// TIA Portal V17 export
// export: Created 2023-03-06T02:05:12.3050921Z, ExportSetting WithDefaults, DisplayName Totally Integrated Automation Portal, DisplayVersion V17 Update 4, DisplayName TIA Portal Openness, DisplayVersion V17 Update 4, DisplayName TIA Portal Version Control Interface, DisplayVersion V17, DisplayName STEP 7 Professional, DisplayVersion V17 Update 4, DisplayName STEP 7 Safety, DisplayVersion V17, DisplayName WinCC Professional, DisplayVersion V17 Update 4
FUNCTION "PCS1 W (PE)" : Void   // FC42, LAD
TITLE = ModBus TCP for PCS Power Electronics
{ S7_Optimized_Access := 'TRUE' }
VERSION : 0.1
// stored: AutoNumber false, IsIECCheckEnabled false, SetENOAutomatically false, UDAEnableTagReadback false
   VAR_TEMP
      rSS1PacRef : Real;
      rSS2PacRef : Real;
      rSS1QacRef : Real;
      rSS2QacRef : Real;
      rSnHalfPE : Real;
   END_VAR
   VAR_TEMP   // added for the SCL form of the ladder/FBD networks
      _w1 : Bool;
      _w2 : Bool;
   END_VAR
BEGIN

REGION Network 1: Function Modbus Client
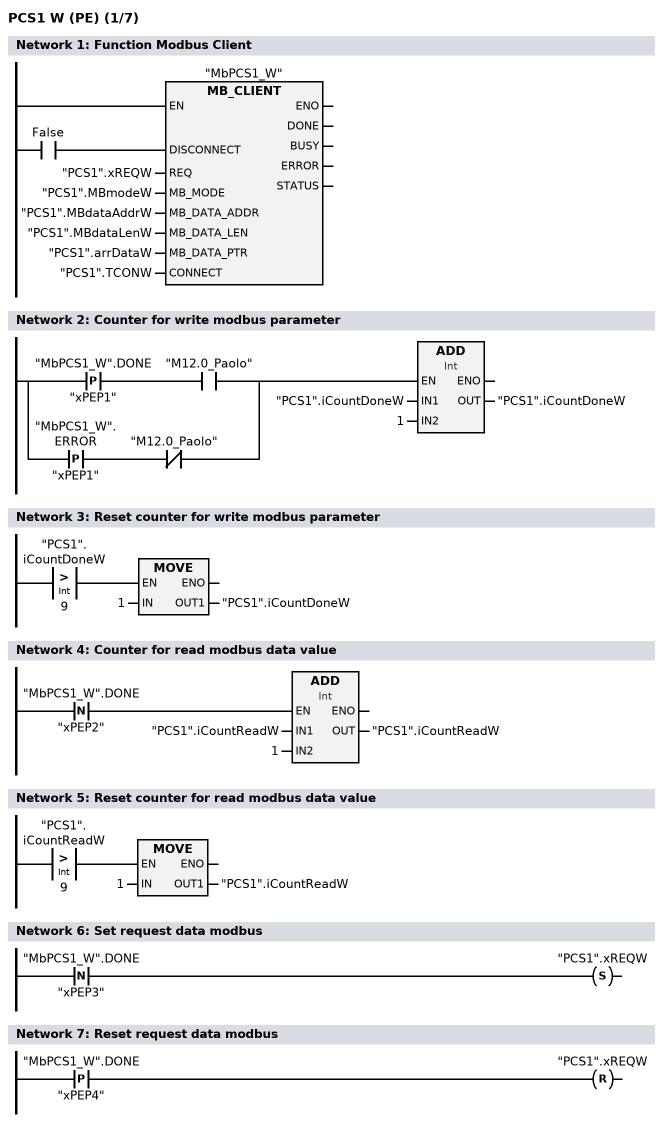
   RUNG wire#powerrail
      "MbPCS1_W".MB_CLIENT(DISCONNECT := wire#w1, REQ := "PCS1".xREQW, MB_MODE := "PCS1".MBmodeW, MB_DATA_ADDR := "PCS1".MBdataAddrW, MB_DATA_LEN := "PCS1".MBdataLenW, MB_DATA_PTR := "PCS1".arrDataW, CONNECT := "PCS1".TCONW, DONE =>, BUSY =>, ERROR =>, STATUS =>)
   END_RUNG
   RUNG wire#powerrail
      Contact( False )
   END_RUNG wire#w1
   // the same network as SCL:
   "MbPCS1_W"(DISCONNECT := False,   // MB_CLIENT
              REQ := "PCS1".xREQW,
              MB_MODE := "PCS1".MBmodeW,
              MB_DATA_ADDR := "PCS1".MBdataAddrW,
              MB_DATA_LEN := "PCS1".MBdataLenW,
              MB_DATA_PTR := "PCS1".arrDataW,
              CONNECT := "PCS1".TCONW);
END_REGION

REGION Network 2: Counter for write modbus parameter
   RUNG wire#powerrail
      P_Contact(operand := "MbPCS1_W".DONE, bit := "xPEP1")
      Contact( "M12.0_Paolo" )
      wire#w1
      { S7_Templates := "SrcType := Int" } Add(in1 := "PCS1".iCountDoneW, in2 := 1, out => "PCS1".iCountDoneW)
   END_RUNG
   RUNG wire#powerrail
      P_Contact(operand := "MbPCS1_W".ERROR, bit := "xPEP1")
      I_Contact( "M12.0_Paolo" )
   END_RUNG wire#w1
   // the same network as SCL:
   #_w1 := "MbPCS1_W".DONE AND NOT "xPEP1";   // rising edge of "MbPCS1_W".DONE
   "xPEP1" := "MbPCS1_W".DONE;
   #_w2 := "MbPCS1_W".ERROR AND NOT "xPEP1";   // rising edge of "MbPCS1_W".ERROR
   "xPEP1" := "MbPCS1_W".ERROR;
   IF (#_w1 AND "M12.0_Paolo") OR (#_w2 AND NOT "M12.0_Paolo") THEN
       "PCS1".iCountDoneW := "PCS1".iCountDoneW + 1;
   END_IF;
END_REGION

REGION Network 3: Reset counter for write modbus parameter
   RUNG wire#powerrail
      { S7_Templates := "SrcType := Int" } GT_Contact(in1 := "PCS1".iCountDoneW, in2 := 9)
      Move(in := 1, out1 => "PCS1".iCountDoneW)
   END_RUNG
   // the same network as SCL:
   IF "PCS1".iCountDoneW > 9 THEN "PCS1".iCountDoneW := 1; END_IF;
END_REGION

REGION Network 4: Counter for read modbus data value
   RUNG wire#powerrail
      N_Contact(operand := "MbPCS1_W".DONE, bit := "xPEP2")
      { S7_Templates := "SrcType := Int" } Add(in1 := "PCS1".iCountReadW, in2 := 1, out => "PCS1".iCountReadW)
   END_RUNG
   // the same network as SCL:
   #_w1 := NOT "MbPCS1_W".DONE AND "xPEP2";   // falling edge of "MbPCS1_W".DONE
   "xPEP2" := "MbPCS1_W".DONE;
   IF #_w1 THEN "PCS1".iCountReadW := "PCS1".iCountReadW + 1; END_IF;
END_REGION

REGION Network 5: Reset counter for read modbus data value
   RUNG wire#powerrail
      { S7_Templates := "SrcType := Int" } GT_Contact(in1 := "PCS1".iCountReadW, in2 := 9)
      Move(in := 1, out1 => "PCS1".iCountReadW)
   END_RUNG
   // the same network as SCL:
   IF "PCS1".iCountReadW > 9 THEN "PCS1".iCountReadW := 1; END_IF;
END_REGION

REGION Network 6: Set request data modbus
   RUNG wire#powerrail
      N_Contact(operand := "MbPCS1_W".DONE, bit := "xPEP3")
      S_Coil( "PCS1".xREQW )
   END_RUNG
   // the same network as SCL:
   #_w1 := NOT "MbPCS1_W".DONE AND "xPEP3";   // falling edge of "MbPCS1_W".DONE
   "xPEP3" := "MbPCS1_W".DONE;
   IF #_w1 THEN "PCS1".xREQW := TRUE; END_IF;
END_REGION

REGION Network 7: Reset request data modbus
   RUNG wire#powerrail
      P_Contact(operand := "MbPCS1_W".DONE, bit := "xPEP4")
      R_Coil( "PCS1".xREQW )
   END_RUNG
   // the same network as SCL:
   #_w1 := "MbPCS1_W".DONE AND NOT "xPEP4";   // rising edge of "MbPCS1_W".DONE
   "xPEP4" := "MbPCS1_W".DONE;
   IF #_w1 THEN "PCS1".xREQW := FALSE; END_IF;
END_REGION

REGION Network 9: Write W_Block1 parameter
   // wUserPswIns
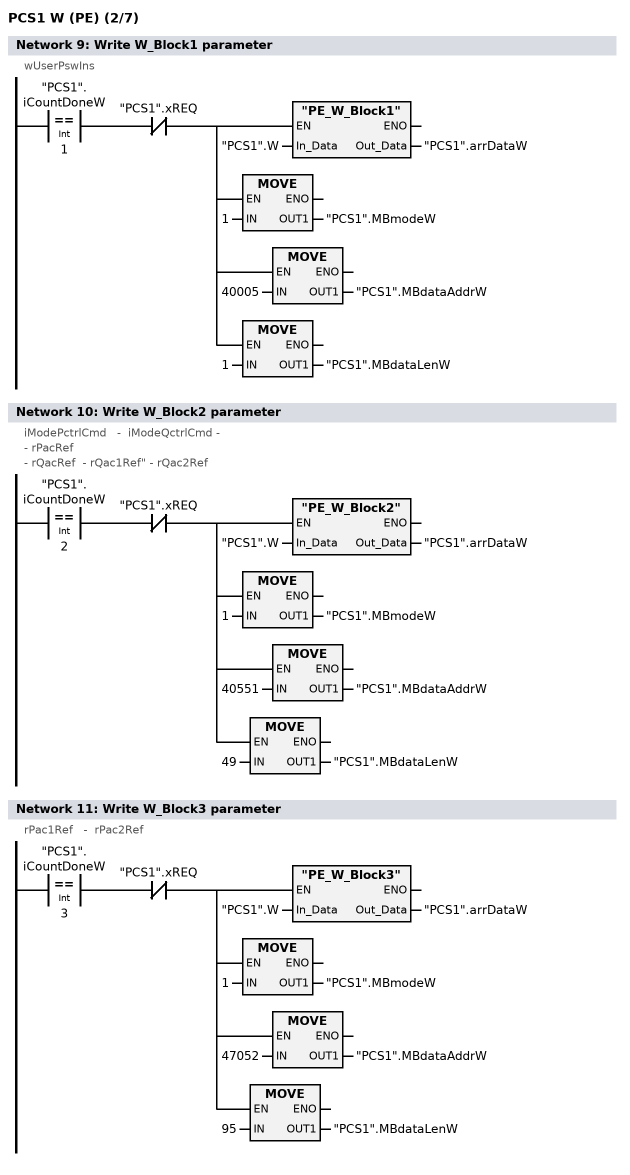
   RUNG wire#powerrail
      { S7_Templates := "SrcType := Int" } EQ_Contact(in1 := "PCS1".iCountDoneW, in2 := 1)
      I_Contact( "PCS1".xREQ )
      wire#w1
      "PE_W_Block1"(In_Data := "PCS1".W, Out_Data => "PCS1".arrDataW)
   END_RUNG
   RUNG wire#w1
      Move(in := 1, out1 => "PCS1".MBmodeW)
   END_RUNG
   RUNG wire#w1
      Move(in := 40005, out1 => "PCS1".MBdataAddrW)
   END_RUNG
   RUNG wire#w1
      Move(in := 1, out1 => "PCS1".MBdataLenW)
   END_RUNG
   // the same network as SCL:
   #_w1 := ("PCS1".iCountDoneW = 1) AND NOT "PCS1".xREQ;
   IF #_w1 THEN
       "PE_W_Block1"(In_Data := "PCS1".W, Out_Data => "PCS1".arrDataW);
       "PCS1".MBmodeW := 1;
       "PCS1".MBdataAddrW := 40005;
       "PCS1".MBdataLenW := 1;
   END_IF;
END_REGION

REGION Network 10: Write W_Block2 parameter
   // iModePctrlCmd   -  iModeQctrlCmd - 
   // - rPacRef 
   // - rQacRef  - rQac1Ref" - rQac2Ref
   RUNG wire#powerrail
      { S7_Templates := "SrcType := Int" } EQ_Contact(in1 := "PCS1".iCountDoneW, in2 := 2)
      I_Contact( "PCS1".xREQ )
      wire#w1
      "PE_W_Block2"(In_Data := "PCS1".W, Out_Data => "PCS1".arrDataW)
   END_RUNG
   RUNG wire#w1
      Move(in := 1, out1 => "PCS1".MBmodeW)
   END_RUNG
   RUNG wire#w1
      Move(in := 40551, out1 => "PCS1".MBdataAddrW)
   END_RUNG
   RUNG wire#w1
      Move(in := 49, out1 => "PCS1".MBdataLenW)
   END_RUNG
   // the same network as SCL:
   #_w1 := ("PCS1".iCountDoneW = 2) AND NOT "PCS1".xREQ;
   IF #_w1 THEN
       "PE_W_Block2"(In_Data := "PCS1".W, Out_Data => "PCS1".arrDataW);
       "PCS1".MBmodeW := 1;
       "PCS1".MBdataAddrW := 40551;
       "PCS1".MBdataLenW := 49;
   END_IF;
END_REGION

REGION Network 11: Write W_Block3 parameter
   // rPac1Ref   -  rPac2Ref
   RUNG wire#powerrail
      { S7_Templates := "SrcType := Int" } EQ_Contact(in1 := "PCS1".iCountDoneW, in2 := 3)
      I_Contact( "PCS1".xREQ )
      wire#w1
      "PE_W_Block3"(In_Data := "PCS1".W, Out_Data => "PCS1".arrDataW)
   END_RUNG
   RUNG wire#w1
      Move(in := 1, out1 => "PCS1".MBmodeW)
   END_RUNG
   RUNG wire#w1
      Move(in := 47052, out1 => "PCS1".MBdataAddrW)
   END_RUNG
   RUNG wire#w1
      Move(in := 95, out1 => "PCS1".MBdataLenW)
   END_RUNG
   // the same network as SCL:
   #_w1 := ("PCS1".iCountDoneW = 3) AND NOT "PCS1".xREQ;
   IF #_w1 THEN
       "PE_W_Block3"(In_Data := "PCS1".W, Out_Data => "PCS1".arrDataW);
       "PCS1".MBmodeW := 1;
       "PCS1".MBdataAddrW := 47052;
       "PCS1".MBdataLenW := 95;
   END_IF;
END_REGION

REGION Network 12: Write Command Start
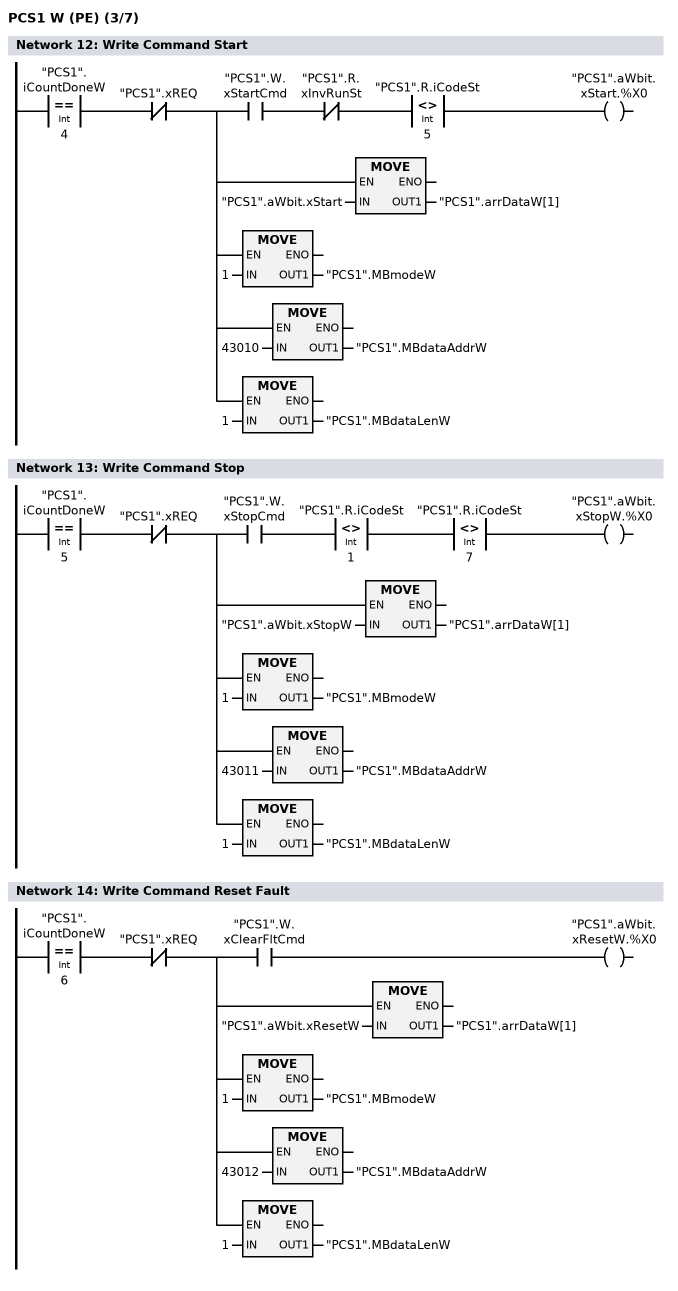
   RUNG wire#powerrail
      { S7_Templates := "SrcType := Int" } EQ_Contact(in1 := "PCS1".iCountDoneW, in2 := 4)
      I_Contact( "PCS1".xREQ )
      wire#w1
      Contact( "PCS1".W.xStartCmd )
      I_Contact( "PCS1".R.xInvRunSt )
      { S7_Templates := "SrcType := Int" } NE_Contact(in1 := "PCS1".R.iCodeSt, in2 := 5)
      Coil( "PCS1".aWbit.xStart.%X0 )
   END_RUNG
   RUNG wire#w1
      Move(in := "PCS1".aWbit.xStart, out1 => "PCS1".arrDataW[1])
   END_RUNG
   RUNG wire#w1
      Move(in := 1, out1 => "PCS1".MBmodeW)
   END_RUNG
   RUNG wire#w1
      Move(in := 43010, out1 => "PCS1".MBdataAddrW)
   END_RUNG
   RUNG wire#w1
      Move(in := 1, out1 => "PCS1".MBdataLenW)
   END_RUNG
   // the same network as SCL:
   #_w1 := ("PCS1".iCountDoneW = 4) AND NOT "PCS1".xREQ;
   "PCS1".aWbit.xStart.%X0 := #_w1 AND "PCS1".W.xStartCmd AND NOT "PCS1".R.xInvRunSt AND ("PCS1".R.iCodeSt <> 5);
   IF #_w1 THEN
       "PCS1".arrDataW[1] := "PCS1".aWbit.xStart;
       "PCS1".MBmodeW := 1;
       "PCS1".MBdataAddrW := 43010;
       "PCS1".MBdataLenW := 1;
   END_IF;
END_REGION

REGION Network 13: Write Command Stop
   RUNG wire#powerrail
      { S7_Templates := "SrcType := Int" } EQ_Contact(in1 := "PCS1".iCountDoneW, in2 := 5)
      I_Contact( "PCS1".xREQ )
      wire#w1
      Contact( "PCS1".W.xStopCmd )
      { S7_Templates := "SrcType := Int" } NE_Contact(in1 := "PCS1".R.iCodeSt, in2 := 1)
      { S7_Templates := "SrcType := Int" } NE_Contact(in1 := "PCS1".R.iCodeSt, in2 := 7)
      Coil( "PCS1".aWbit.xStopW.%X0 )
   END_RUNG
   RUNG wire#w1
      Move(in := "PCS1".aWbit.xStopW, out1 => "PCS1".arrDataW[1])
   END_RUNG
   RUNG wire#w1
      Move(in := 1, out1 => "PCS1".MBmodeW)
   END_RUNG
   RUNG wire#w1
      Move(in := 43011, out1 => "PCS1".MBdataAddrW)
   END_RUNG
   RUNG wire#w1
      Move(in := 1, out1 => "PCS1".MBdataLenW)
   END_RUNG
   // the same network as SCL:
   #_w1 := ("PCS1".iCountDoneW = 5) AND NOT "PCS1".xREQ;
   "PCS1".aWbit.xStopW.%X0 := #_w1 AND "PCS1".W.xStopCmd AND ("PCS1".R.iCodeSt <> 1) AND ("PCS1".R.iCodeSt <> 7);
   IF #_w1 THEN
       "PCS1".arrDataW[1] := "PCS1".aWbit.xStopW;
       "PCS1".MBmodeW := 1;
       "PCS1".MBdataAddrW := 43011;
       "PCS1".MBdataLenW := 1;
   END_IF;
END_REGION

REGION Network 14: Write Command Reset Fault
   RUNG wire#powerrail
      { S7_Templates := "SrcType := Int" } EQ_Contact(in1 := "PCS1".iCountDoneW, in2 := 6)
      I_Contact( "PCS1".xREQ )
      wire#w1
      Contact( "PCS1".W.xClearFltCmd )
      Coil( "PCS1".aWbit.xResetW.%X0 )
   END_RUNG
   RUNG wire#w1
      Move(in := "PCS1".aWbit.xResetW, out1 => "PCS1".arrDataW[1])
   END_RUNG
   RUNG wire#w1
      Move(in := 1, out1 => "PCS1".MBmodeW)
   END_RUNG
   RUNG wire#w1
      Move(in := 43012, out1 => "PCS1".MBdataAddrW)
   END_RUNG
   RUNG wire#w1
      Move(in := 1, out1 => "PCS1".MBdataLenW)
   END_RUNG
   // the same network as SCL:
   #_w1 := ("PCS1".iCountDoneW = 6) AND NOT "PCS1".xREQ;
   "PCS1".aWbit.xResetW.%X0 := #_w1 AND "PCS1".W.xClearFltCmd;
   IF #_w1 THEN
       "PCS1".arrDataW[1] := "PCS1".aWbit.xResetW;
       "PCS1".MBmodeW := 1;
       "PCS1".MBdataAddrW := 43012;
       "PCS1".MBdataLenW := 1;
   END_IF;
END_REGION

REGION Network 15: Write Command Enable Start/Stop
   // Con versione vecchia si usava solo questo registro per marcia ed arresto.
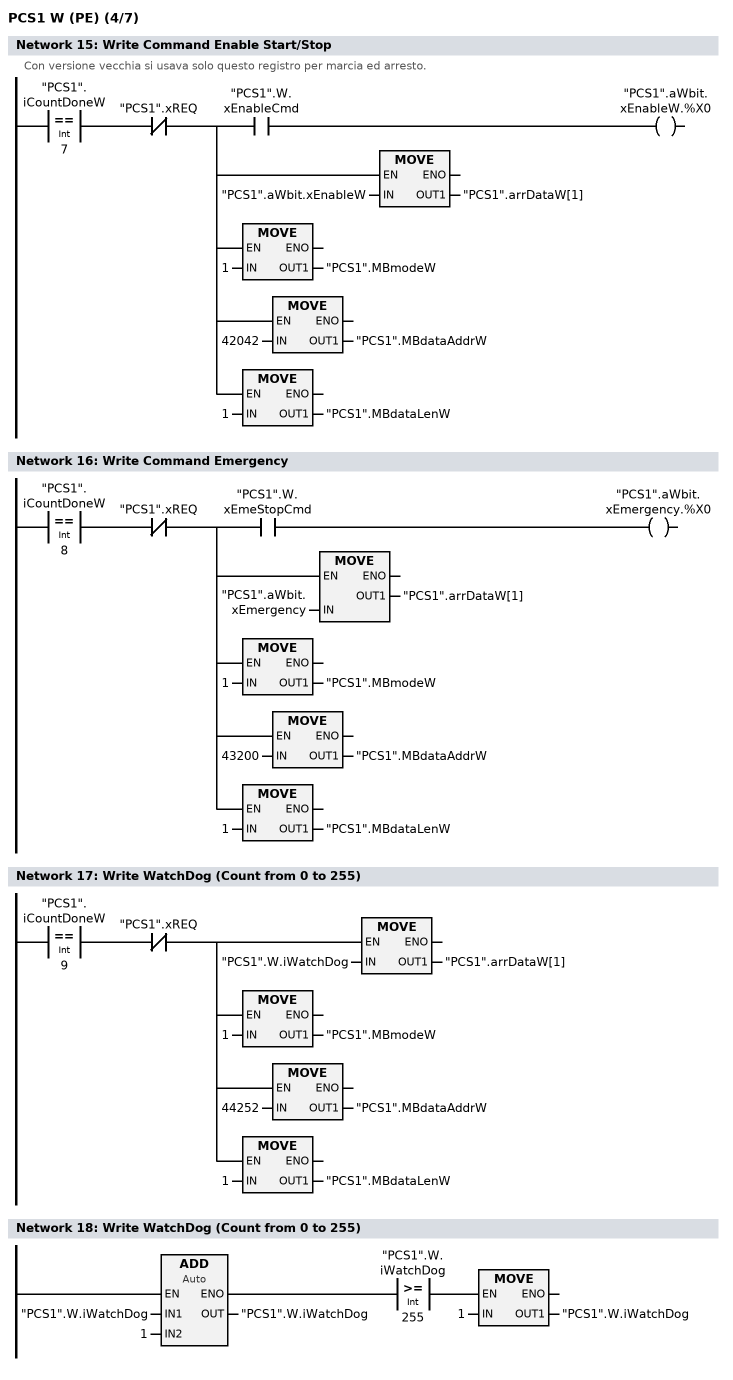
   RUNG wire#powerrail
      { S7_Templates := "SrcType := Int" } EQ_Contact(in1 := "PCS1".iCountDoneW, in2 := 7)
      I_Contact( "PCS1".xREQ )
      wire#w1
      Contact( "PCS1".W.xEnableCmd )
      Coil( "PCS1".aWbit.xEnableW.%X0 )
   END_RUNG
   RUNG wire#w1
      Move(in := "PCS1".aWbit.xEnableW, out1 => "PCS1".arrDataW[1])
   END_RUNG
   RUNG wire#w1
      Move(in := 1, out1 => "PCS1".MBmodeW)
   END_RUNG
   RUNG wire#w1
      Move(in := 42042, out1 => "PCS1".MBdataAddrW)
   END_RUNG
   RUNG wire#w1
      Move(in := 1, out1 => "PCS1".MBdataLenW)
   END_RUNG
   // the same network as SCL:
   #_w1 := ("PCS1".iCountDoneW = 7) AND NOT "PCS1".xREQ;
   "PCS1".aWbit.xEnableW.%X0 := #_w1 AND "PCS1".W.xEnableCmd;
   IF #_w1 THEN
       "PCS1".arrDataW[1] := "PCS1".aWbit.xEnableW;
       "PCS1".MBmodeW := 1;
       "PCS1".MBdataAddrW := 42042;
       "PCS1".MBdataLenW := 1;
   END_IF;
END_REGION

REGION Network 16: Write Command Emergency
   RUNG wire#powerrail
      { S7_Templates := "SrcType := Int" } EQ_Contact(in1 := "PCS1".iCountDoneW, in2 := 8)
      I_Contact( "PCS1".xREQ )
      wire#w1
      Contact( "PCS1".W.xEmeStopCmd )
      Coil( "PCS1".aWbit.xEmergency.%X0 )
   END_RUNG
   RUNG wire#w1
      Move(in := "PCS1".aWbit.xEmergency, out1 => "PCS1".arrDataW[1])
   END_RUNG
   RUNG wire#w1
      Move(in := 1, out1 => "PCS1".MBmodeW)
   END_RUNG
   RUNG wire#w1
      Move(in := 43200, out1 => "PCS1".MBdataAddrW)
   END_RUNG
   RUNG wire#w1
      Move(in := 1, out1 => "PCS1".MBdataLenW)
   END_RUNG
   // the same network as SCL:
   #_w1 := ("PCS1".iCountDoneW = 8) AND NOT "PCS1".xREQ;
   "PCS1".aWbit.xEmergency.%X0 := #_w1 AND "PCS1".W.xEmeStopCmd;
   IF #_w1 THEN
       "PCS1".arrDataW[1] := "PCS1".aWbit.xEmergency;
       "PCS1".MBmodeW := 1;
       "PCS1".MBdataAddrW := 43200;
       "PCS1".MBdataLenW := 1;
   END_IF;
END_REGION

REGION Network 17: Write WatchDog (Count from 0 to 255)
   RUNG wire#powerrail
      { S7_Templates := "SrcType := Int" } EQ_Contact(in1 := "PCS1".iCountDoneW, in2 := 9)
      I_Contact( "PCS1".xREQ )
      wire#w1
      Move(in := "PCS1".W.iWatchDog, out1 => "PCS1".arrDataW[1])
   END_RUNG
   RUNG wire#w1
      Move(in := 1, out1 => "PCS1".MBmodeW)
   END_RUNG
   RUNG wire#w1
      Move(in := 44252, out1 => "PCS1".MBdataAddrW)
   END_RUNG
   RUNG wire#w1
      Move(in := 1, out1 => "PCS1".MBdataLenW)
   END_RUNG
   // the same network as SCL:
   IF ("PCS1".iCountDoneW = 9) AND NOT "PCS1".xREQ THEN
       "PCS1".arrDataW[1] := "PCS1".W.iWatchDog;
       "PCS1".MBmodeW := 1;
       "PCS1".MBdataAddrW := 44252;
       "PCS1".MBdataLenW := 1;
   END_IF;
END_REGION

REGION Network 18: Write WatchDog (Count from 0 to 255)
   RUNG wire#powerrail
      Add(in1 := "PCS1".W.iWatchDog, in2 := 1, out => "PCS1".W.iWatchDog)
      { S7_Templates := "SrcType := Int" } GE_Contact(in1 := "PCS1".W.iWatchDog, in2 := 255)
      Move(in := 1, out1 => "PCS1".W.iWatchDog)
   END_RUNG
   // the same network as SCL:
   "PCS1".W.iWatchDog := "PCS1".W.iWatchDog + 1;
   IF "PCS1".W.iWatchDog >= 255 THEN "PCS1".W.iWatchDog := 1; END_IF;
END_REGION

REGION Network 20: 43010
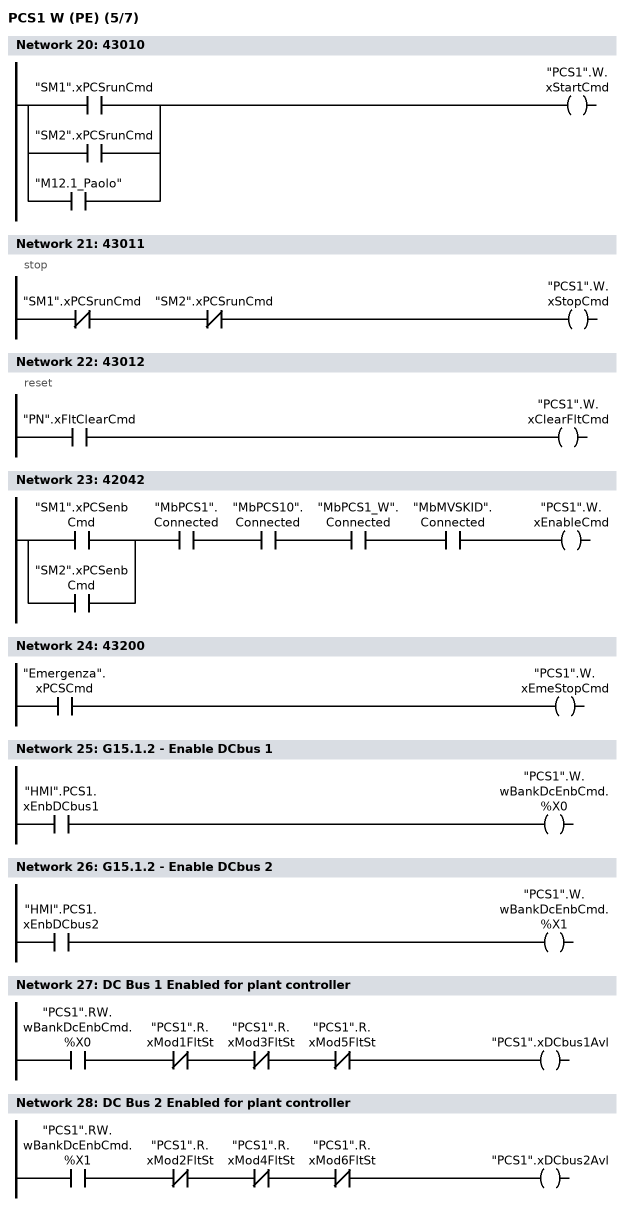
   RUNG wire#powerrail
      Contact( "SM1".xPCSrunCmd )
      wire#w1
      Coil( "PCS1".W.xStartCmd )
   END_RUNG
   RUNG wire#powerrail
      Contact( "SM2".xPCSrunCmd )
   END_RUNG wire#w1
   RUNG wire#powerrail
      Contact( "M12.1_Paolo" )
   END_RUNG wire#w1
   // the same network as SCL:
   "PCS1".W.xStartCmd := "SM1".xPCSrunCmd OR "SM2".xPCSrunCmd OR "M12.1_Paolo";
END_REGION

REGION Network 21: 43011
   // stop
   RUNG wire#powerrail
      I_Contact( "SM1".xPCSrunCmd )
      I_Contact( "SM2".xPCSrunCmd )
      Coil( "PCS1".W.xStopCmd )
   END_RUNG
   // the same network as SCL:
   "PCS1".W.xStopCmd := NOT "SM1".xPCSrunCmd AND NOT "SM2".xPCSrunCmd;
END_REGION

REGION Network 22: 43012
   // reset
   RUNG wire#powerrail
      Contact( "PN".xFltClearCmd )
      Coil( "PCS1".W.xClearFltCmd )
   END_RUNG
   // the same network as SCL:
   "PCS1".W.xClearFltCmd := "PN".xFltClearCmd;
END_REGION

REGION Network 23: 42042
   RUNG wire#powerrail
      Contact( "SM1".xPCSenbCmd )
      wire#w1
      Contact( "MbPCS1".Connected )
      Contact( "MbPCS10".Connected )
      Contact( "MbPCS1_W".Connected )
      Contact( "MbMVSKID".Connected )
      Coil( "PCS1".W.xEnableCmd )
   END_RUNG
   RUNG wire#powerrail
      Contact( "SM2".xPCSenbCmd )
   END_RUNG wire#w1
   // the same network as SCL:
   "PCS1".W.xEnableCmd := ("SM1".xPCSenbCmd OR "SM2".xPCSenbCmd) AND "MbPCS1".Connected AND "MbPCS10".Connected AND "MbPCS1_W".Connected AND "MbMVSKID".Connected;
END_REGION

REGION Network 24: 43200
   RUNG wire#powerrail
      Contact( "Emergenza".xPCSCmd )
      Coil( "PCS1".W.xEmeStopCmd )
   END_RUNG
   // the same network as SCL:
   "PCS1".W.xEmeStopCmd := "Emergenza".xPCSCmd;
END_REGION

REGION Network 25: G15.1.2 - Enable DCbus 1
   RUNG wire#powerrail
      Contact( "HMI".PCS1.xEnbDCbus1 )
      Coil( "PCS1".W.wBankDcEnbCmd.%X0 )
   END_RUNG
   // the same network as SCL:
   "PCS1".W.wBankDcEnbCmd.%X0 := "HMI".PCS1.xEnbDCbus1;
END_REGION

REGION Network 26: G15.1.2 - Enable DCbus 2
   RUNG wire#powerrail
      Contact( "HMI".PCS1.xEnbDCbus2 )
      Coil( "PCS1".W.wBankDcEnbCmd.%X1 )
   END_RUNG
   // the same network as SCL:
   "PCS1".W.wBankDcEnbCmd.%X1 := "HMI".PCS1.xEnbDCbus2;
END_REGION

REGION Network 27: DC Bus 1 Enabled for plant controller
   RUNG wire#powerrail
      Contact( "PCS1".RW.wBankDcEnbCmd.%X0 )
      I_Contact( "PCS1".R.xMod1FltSt )
      I_Contact( "PCS1".R.xMod3FltSt )
      I_Contact( "PCS1".R.xMod5FltSt )
      Coil( "PCS1".xDCbus1Avl )
   END_RUNG
   // the same network as SCL:
   "PCS1".xDCbus1Avl := "PCS1".RW.wBankDcEnbCmd.%X0 AND NOT "PCS1".R.xMod1FltSt AND NOT "PCS1".R.xMod3FltSt AND NOT "PCS1".R.xMod5FltSt;
END_REGION

REGION Network 28: DC Bus 2 Enabled for plant controller
   RUNG wire#powerrail
      Contact( "PCS1".RW.wBankDcEnbCmd.%X1 )
      I_Contact( "PCS1".R.xMod2FltSt )
      I_Contact( "PCS1".R.xMod4FltSt )
      I_Contact( "PCS1".R.xMod6FltSt )
      Coil( "PCS1".xDCbus2Avl )
   END_RUNG
   // the same network as SCL:
   "PCS1".xDCbus2Avl := "PCS1".RW.wBankDcEnbCmd.%X1 AND NOT "PCS1".R.xMod2FltSt AND NOT "PCS1".R.xMod4FltSt AND NOT "PCS1".R.xMod6FltSt;
END_REGION

REGION Network 30: Active Power local reference for PE with 2 DC Bus
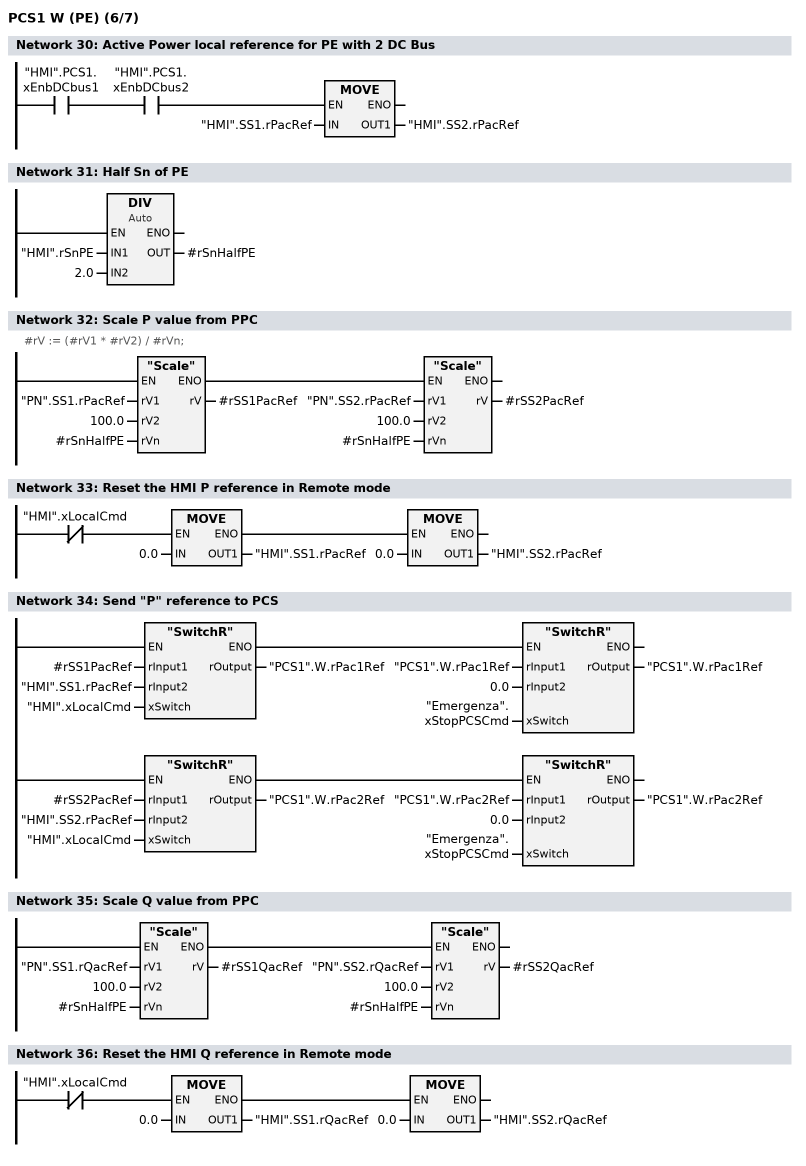
   RUNG wire#powerrail
      Contact( "HMI".PCS1.xEnbDCbus1 )
      Contact( "HMI".PCS1.xEnbDCbus2 )
      Move(in := "HMI".SS1.rPacRef, out1 => "HMI".SS2.rPacRef)
   END_RUNG
   // the same network as SCL:
   IF "HMI".PCS1.xEnbDCbus1 AND "HMI".PCS1.xEnbDCbus2 THEN "HMI".SS2.rPacRef := "HMI".SS1.rPacRef; END_IF;
END_REGION

REGION Network 31: Half Sn of PE
   RUNG wire#powerrail
      Div(in1 := "HMI".rSnPE, in2 := 2.0, out => #rSnHalfPE)
   END_RUNG
   // the same network as SCL:
   #rSnHalfPE := "HMI".rSnPE / 2.0;
END_REGION

REGION Network 32: Scale P value from PPC
   // #rV := (#rV1 * #rV2) / #rVn;
   RUNG wire#powerrail
      "Scale"(rV1 := "PN".SS1.rPacRef, rV2 := 100.0, rVn := #rSnHalfPE, rV => #rSS1PacRef)
      "Scale"(rV1 := "PN".SS2.rPacRef, rV2 := 100.0, rVn := #rSnHalfPE, rV => #rSS2PacRef)
   END_RUNG
   // the same network as SCL:
   "Scale"(rV1 := "PN".SS1.rPacRef, rV2 := 100.0, rVn := #rSnHalfPE, rV => #rSS1PacRef, ENO => #_w1);
   IF #_w1 THEN "Scale"(rV1 := "PN".SS2.rPacRef, rV2 := 100.0, rVn := #rSnHalfPE, rV => #rSS2PacRef); END_IF;
END_REGION

REGION Network 33: Reset the HMI P reference in Remote mode
   RUNG wire#powerrail
      I_Contact( "HMI".xLocalCmd )
      Move(in := 0.0, out1 => "HMI".SS1.rPacRef)
      Move(in := 0.0, out1 => "HMI".SS2.rPacRef)
   END_RUNG
   // the same network as SCL:
   IF NOT "HMI".xLocalCmd THEN
       "HMI".SS1.rPacRef := 0.0;
       "HMI".SS2.rPacRef := 0.0;
   END_IF;
END_REGION

REGION Network 34: Send "P" reference to PCS
   RUNG wire#powerrail
      "SwitchR"(rInput1 := #rSS1PacRef, rInput2 := "HMI".SS1.rPacRef, xSwitch := "HMI".xLocalCmd, rOutput => "PCS1".W.rPac1Ref)
      "SwitchR"(rInput1 := "PCS1".W.rPac1Ref, rInput2 := 0.0, xSwitch := "Emergenza".xStopPCSCmd, rOutput => "PCS1".W.rPac1Ref)
   END_RUNG
   RUNG wire#powerrail
      "SwitchR"(rInput1 := #rSS2PacRef, rInput2 := "HMI".SS2.rPacRef, xSwitch := "HMI".xLocalCmd, rOutput => "PCS1".W.rPac2Ref)
      "SwitchR"(rInput1 := "PCS1".W.rPac2Ref, rInput2 := 0.0, xSwitch := "Emergenza".xStopPCSCmd, rOutput => "PCS1".W.rPac2Ref)
   END_RUNG
   // the same network as SCL:
   "SwitchR"(rInput1 := #rSS1PacRef,
             rInput2 := "HMI".SS1.rPacRef,
             xSwitch := "HMI".xLocalCmd,
             rOutput => "PCS1".W.rPac1Ref,
             ENO => #_w1);
   IF #_w1 THEN
       "SwitchR"(rInput1 := "PCS1".W.rPac1Ref,
                 rInput2 := 0.0,
                 xSwitch := "Emergenza".xStopPCSCmd,
                 rOutput => "PCS1".W.rPac1Ref);
   END_IF;
   "SwitchR"(rInput1 := #rSS2PacRef,
             rInput2 := "HMI".SS2.rPacRef,
             xSwitch := "HMI".xLocalCmd,
             rOutput => "PCS1".W.rPac2Ref,
             ENO => #_w2);
   IF #_w2 THEN
       "SwitchR"(rInput1 := "PCS1".W.rPac2Ref,
                 rInput2 := 0.0,
                 xSwitch := "Emergenza".xStopPCSCmd,
                 rOutput => "PCS1".W.rPac2Ref);
   END_IF;
END_REGION

REGION Network 35: Scale Q value from PPC
   RUNG wire#powerrail
      "Scale"(rV1 := "PN".SS1.rQacRef, rV2 := 100.0, rVn := #rSnHalfPE, rV => #rSS1QacRef)
      "Scale"(rV1 := "PN".SS2.rQacRef, rV2 := 100.0, rVn := #rSnHalfPE, rV => #rSS2QacRef)
   END_RUNG
   // the same network as SCL:
   "Scale"(rV1 := "PN".SS1.rQacRef, rV2 := 100.0, rVn := #rSnHalfPE, rV => #rSS1QacRef, ENO => #_w1);
   IF #_w1 THEN "Scale"(rV1 := "PN".SS2.rQacRef, rV2 := 100.0, rVn := #rSnHalfPE, rV => #rSS2QacRef); END_IF;
END_REGION

REGION Network 36: Reset the HMI Q reference in Remote mode
   RUNG wire#powerrail
      I_Contact( "HMI".xLocalCmd )
      Move(in := 0.0, out1 => "HMI".SS1.rQacRef)
      Move(in := 0.0, out1 => "HMI".SS2.rQacRef)
   END_RUNG
   // the same network as SCL:
   IF NOT "HMI".xLocalCmd THEN
       "HMI".SS1.rQacRef := 0.0;
       "HMI".SS2.rQacRef := 0.0;
   END_IF;
END_REGION

REGION Network 37: Send "Q" reference to PCS
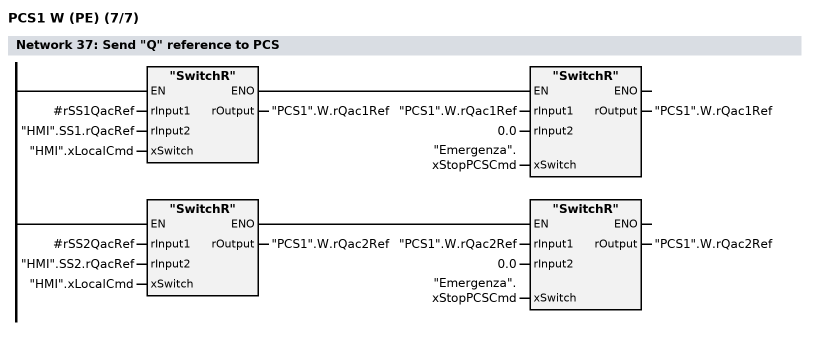
   RUNG wire#powerrail
      "SwitchR"(rInput1 := #rSS1QacRef, rInput2 := "HMI".SS1.rQacRef, xSwitch := "HMI".xLocalCmd, rOutput => "PCS1".W.rQac1Ref)
      "SwitchR"(rInput1 := "PCS1".W.rQac1Ref, rInput2 := 0.0, xSwitch := "Emergenza".xStopPCSCmd, rOutput => "PCS1".W.rQac1Ref)
   END_RUNG
   RUNG wire#powerrail
      "SwitchR"(rInput1 := #rSS2QacRef, rInput2 := "HMI".SS2.rQacRef, xSwitch := "HMI".xLocalCmd, rOutput => "PCS1".W.rQac2Ref)
      "SwitchR"(rInput1 := "PCS1".W.rQac2Ref, rInput2 := 0.0, xSwitch := "Emergenza".xStopPCSCmd, rOutput => "PCS1".W.rQac2Ref)
   END_RUNG
   // the same network as SCL:
   "SwitchR"(rInput1 := #rSS1QacRef,
             rInput2 := "HMI".SS1.rQacRef,
             xSwitch := "HMI".xLocalCmd,
             rOutput => "PCS1".W.rQac1Ref,
             ENO => #_w1);
   IF #_w1 THEN
       "SwitchR"(rInput1 := "PCS1".W.rQac1Ref,
                 rInput2 := 0.0,
                 xSwitch := "Emergenza".xStopPCSCmd,
                 rOutput => "PCS1".W.rQac1Ref);
   END_IF;
   "SwitchR"(rInput1 := #rSS2QacRef,
             rInput2 := "HMI".SS2.rQacRef,
             xSwitch := "HMI".xLocalCmd,
             rOutput => "PCS1".W.rQac2Ref,
             ENO => #_w2);
   IF #_w2 THEN
       "SwitchR"(rInput1 := "PCS1".W.rQac2Ref,
                 rInput2 := 0.0,
                 xSwitch := "Emergenza".xStopPCSCmd,
                 rOutput => "PCS1".W.rQac2Ref);
   END_IF;
END_REGION
END_FUNCTION
